// TIA Portal V18 export
FUNCTION "AIS" : Void   // FC13, LAD
{ S7_Optimized_Access := 'TRUE' }
// stored: SetENOAutomatically false
   VAR_INPUT
      Float_Input : Int;
      Hi_Lmt : Real;
      Low_Lmt : Real;
      K1 : Real;
      K2 : Real;
   END_VAR
   VAR_OUTPUT
      Out_Scale : Real;
   END_VAR
   VAR_TEMP
      Real_1 : Real;
      Real_2 : Real;
      Real_3 : Real;
      Real_4 : Real;
      Float_Real_IN : Real;
   END_VAR
BEGIN

REGION Network 1
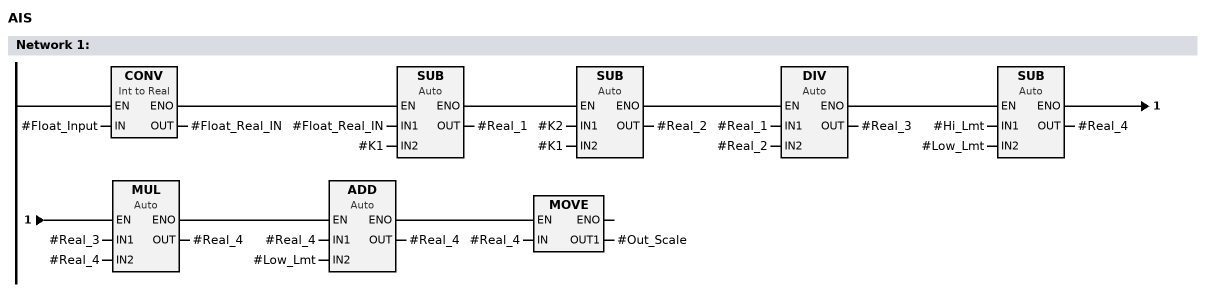
   RUNG wire#powerrail
      { S7_Templates := "[SrcType := Int, DestType := Real]" } Convert(in := #Float_Input, out => #Float_Real_IN)
      Sub(in1 := #Float_Real_IN, in2 := #K1, out => #Real_1)
      Sub(in1 := #K2, in2 := #K1, out => #Real_2)
      Div(in1 := #Real_1, in2 := #Real_2, out => #Real_3)
      Sub(in1 := #Hi_Lmt, in2 := #Low_Lmt, out => #Real_4)
      Mul(in1 := #Real_3, in2 := #Real_4, out => #Real_4)
      Add(in1 := #Real_4, in2 := #Low_Lmt, out => #Real_4)
      Move(in := #Real_4, out1 => #Out_Scale)
   END_RUNG
   // the same network as SCL:
   #Float_Real_IN := INT_TO_REAL(#Float_Input);
   #Real_1 := #Float_Real_IN - #K1;
   #Real_2 := #K2 - #K1;
   #Real_3 := #Real_1 / #Real_2;
   #Real_4 := #Hi_Lmt - #Low_Lmt;
   #Real_4 := #Real_3 * #Real_4;
   #Real_4 := #Real_4 + #Low_Lmt;
   #Out_Scale := #Real_4;
END_REGION
END_FUNCTION
